PROGRAM Prg_FastCall

Prg.FastCall();

END_PROGRAM

(* stored: Version 1.1.0.1
   POU Prg_FastCall: Id {1b0681f2-6f71-433c-9374-8e11a4d42798}, SpecialFunc None *)
